KUKA KRL program: Sps4.sub

&ACCESS RV
&PARAM TPVW_VERSION=8.3.17
DEF  SPS4 ( )
; FOLD ;%{H} %MKUKATPVW
;Init part of vw_usr_s
VW_USR_S (#USR_INIT_SUB4)

LOOP
;Freilaufende SPS
MAKROSUBMIT4()

WAIT FOR NOT $POWER_FAIL
ENDLOOP
END
;ENDFOLD
